// SIMATIC S7-200 SMART project (STEP 7-Micro/WIN SMART), CPU SR40

ORGANIZATION_BLOCK 主程序:OB1
TITLE=
BEGIN
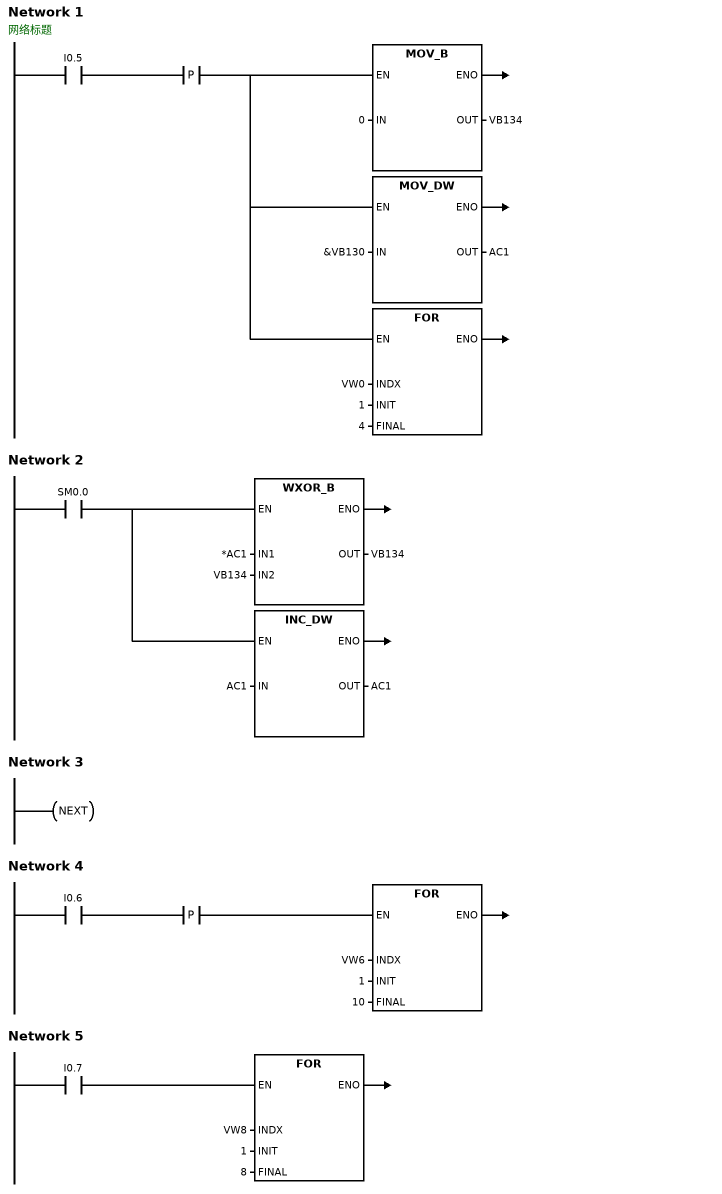
Network 1
// 网络标题
// 在I0.5的上升沿
// 清累加器0
// 累加器1（存储区指针）指向VB10
// 循环开始
LD     I0.5
EU
MOVB   0, VB134
MOVD   &VB130, AC1
FOR    VW0, 1, 4
Network 2
// 字节异或
// 指针AC1的值加1，指向下一个变量存储器字节
LD     SM0.0
XORB   *AC1, VB134
INCD   AC1
Network 3
// 循环结束
NEXT
Network 4
LD     I0.6
EU
FOR    VW6, 1, 10
Network 5
LD     I0.7
FOR    VW8, 1, 8
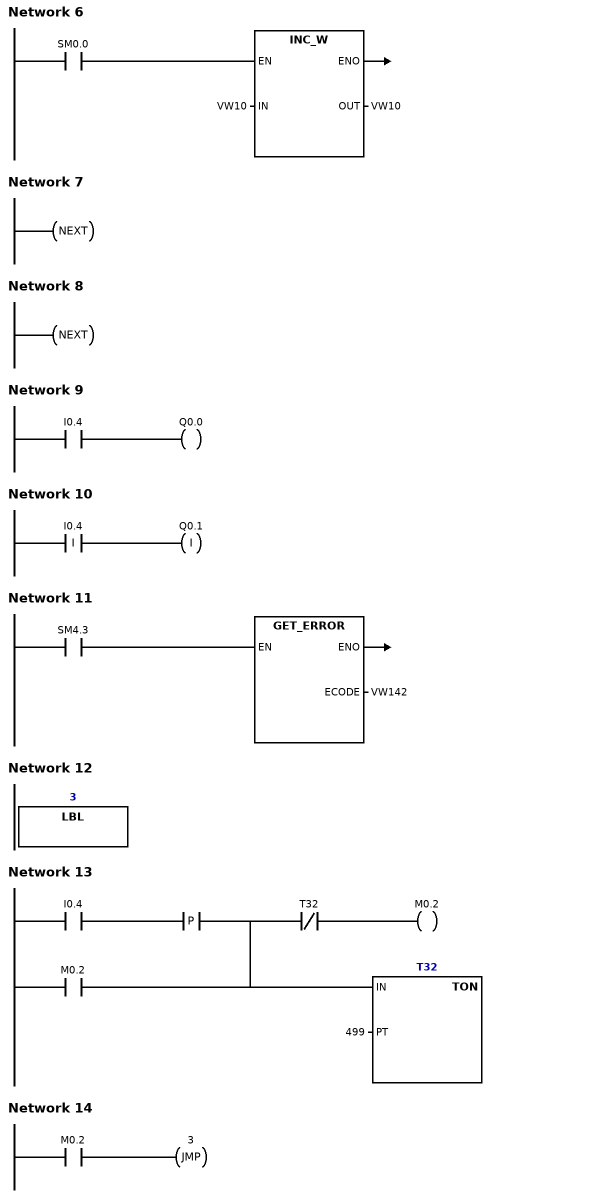
Network 6
LD     SM0.0
INCW   VW10
Network 7
NEXT
Network 8
NEXT
Network 9
LD     I0.4
=      Q0.0
Network 10
LDI    I0.4
=I     Q0.1
Network 11
LD     SM4.3
GERR   VW142
Network 12
LBL    3
Network 13
// (network saved uncompiled; LAD cells follow)
// row 0: c0 -| |- I0.4  c1 -|P|-  v  c2 -|/|- T32  c3 -( ) M0.2
// row 1: c0 -| |- M0.2  c1 -- ^  c2 --  c3 [TON T32 IN:=power@row1, PT:=499]
// row 2: c3 [box]
Network 14
LD     M0.2
JMP    3
END_ORGANIZATION_BLOCK
